Staubli VAL3: power.pgx

public program power(num nPower (dimensions=1))
begin
  //0  to disable power
  //1  to enable power
  switch nPower
    case 0
      disablePower()
    break
    case 1
      enablePower()
    break
    default
      logMsg("power: argumento invalido"+chr(nPower))
    break
  endSwitch
end
